RoboDK station: SETUP Fresas.rdk

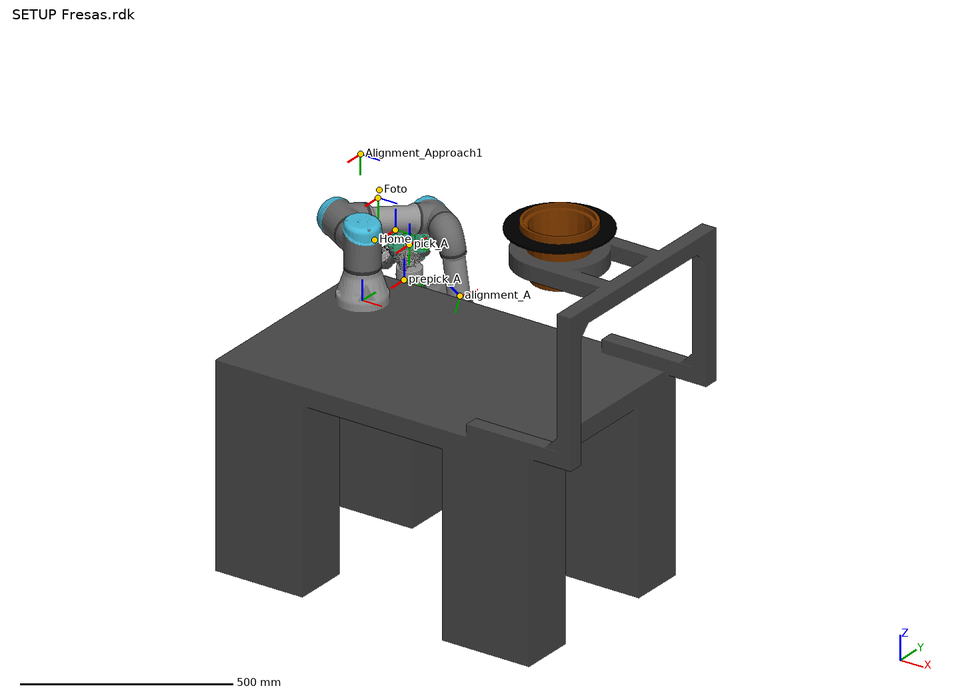
[picture v0: the station drawn from its stored meshes, robots at their saved joint values, targets as dots, program paths as lines]
Station SETUP Fresas (saved by RoboDK 5.9.2). Poses are relative to the parent item; angles as X-Y-Z fixed-axis rotations.
Station parameters (name, value as stored): RECORD_READY, 1, RECORD_ACKNOWLEDGE, 0, CollisionFreeMoveJ, None, CollisionFreeMoveL, None, PathPlanningMaxTime, 5000, PathPlanningMaxIterations, 1000
  - object Mesa SetUp v1 at (600, -20, 0) mm, size 900 x 600 x 550 mm, geometry from Mesa SetUp v1.step
  - frame UR3e Base at (700, 440, 50) mm
    - robot UR3e: 6 axes, payload 3 kg, reach 500 mm, repeatability 0.03 mm, weight 11 kg
        modified DH rows (alpha deg, a mm, theta deg, d mm): 0, 0, 0, 151.9; 90, 0, 180, 0; 0, 243.55, 0, 0; 0, 213.2, 0, 131.05; -90, 0, 0, 85.35; 90, 0, 180, 92.1
        joint limits [-360, -180, -360, -360, -360, -360] to [360, 20, 360, 360, 360, 360]; home [0, -90, -90, 0, 90, 0]; saved at [239.705, 9.056, 73.773, 7.171, -90, -59.705]
      - tool grMK2_betaMK2_asm v6, TCP at (0, 0, 57) mm, size 118.1 x 111.3 x 125.7 mm
      - tool Realsense RGB, TCP at (-11.08, -53.4, 24.76) mm, rotated rx -10 ry 0 rz 0 deg
    - target Home (joint target) at (127.85, -131.05, 246.35) mm, rotated rx -180 ry 0 rz -180 deg; joints [0, -90, -90, 90, -90, -90] of UR3e
    - target Foto (joint target) at (140.09, -131.05, 380) mm, rotated rx -80 ry 0 rz -90 deg; joints [0, -32.82, -150.904, 13.724, 90, 0] of UR3e
    - frame Prepick_plane at (200, -150, 300) mm, rotated rx 0 ry 0 rz -90 deg
      - target Prepick_plane (joint target) at (0, 0, 0) mm; joints [-5.255, -119.46, -148.452, -2.088, -90, -174.745] of UR3e
    - frame Alignment_Approach1 at (100, -150, 470) mm, rotated rx -90 ry 0 rz -90 deg
      - target Alignment_Approach1 (joint target) at (0, 0, 0) mm; joints [15.744, -17.994, -114.376, -47.63, 74.256, 0] of UR3e
    - frame Alignment_Approach2 at (150, -150, 370) mm, rotated rx -90 ry 0 rz -90 deg
      - target Alignment_Approach2 (Cartesian target) at (0, 0, 0) mm; joints [29.458, -1.123, -141.988, -36.888, 60.542, 0] of UR3e
    - target alignment_A (Cartesian target) at (144.6, 193.87, -25.91) mm, rotated rx -70.14 ry 0.6 rz 76.53 deg; joints [60.185, -57.99, -37.957, -95.541, -60.683, 5.683] of UR3e
    - frame alignment_A_frame at (144.6, 193.87, -25.91) mm, rotated rx -70.14 ry 0.6 rz 76.53 deg
    - target prepick_A (Cartesian target) at (-38.34, 226.05, -47.38) mm, rotated rx 0 ry 0 rz -90 deg; joints [60.185, -57.99, -37.957, -95.541, -60.683, 5.683] of UR3e
    - frame prepick_A_frame at (-38.34, 226.05, -47.38) mm, rotated rx 0 ry 0 rz -90 deg
    - target pick_A (Cartesian target) at (-21.45, 223.06, 51.13) mm, rotated rx 0 ry 0 rz -90 deg; joints [60.185, -57.99, -37.957, -95.541, -60.683, 5.683] of UR3e
    - frame pick_A_frame at (-21.45, 223.06, 51.13) mm, rotated rx 0 ry 0 rz -90 deg
    - target post_pick_detach_A (Cartesian target) at (-21.45, 223.06, 51.13) mm, rotated rx -90.14 ry 0.6 rz 76.53 deg; joints [239.705, 9.056, 73.773, 7.171, -90, -59.705] of UR3e
    - frame post_pick_detach_A_frame at (-21.45, 223.06, 51.13) mm, rotated rx -90.14 ry 0.6 rz 76.53 deg
  - object Set Up Fresas YEA v3 at (1570, 280, 60) mm, rotated rx 90 ry 0 rz 180 deg, size 373.6 x 472 x 595 mm, geometry from Set Up Fresas YEA v3.step
  - Python program Giro Brida (listed below)
  - Python program Giro colisiones (listed below)
  - Python program Prog6 (listed below)
  - Python program Hand_Eye_acquisition (listed below)
  - Python program Camera_Live_Stream (listed below)
  - Python program Camera_calibration (listed below)
  - Python program Hand_Eye_calibration (listed below)
  - camera Cámara1

--- Python program Giro Brida ---
from robolink import *    # API de RoboDK
from robodk import *      # Funciones matemáticas
import time
import math
import copy
import sys

# Conexión a RoboDK
RDK = Robolink()

# Intentar seleccionar el robot (usa nombre o el robot activo si '' )
robot = RDK.Item('UR3e', ITEM_TYPE_ROBOT)
if not robot.Valid():
    robot = RDK.Item('', ITEM_TYPE_ROBOT)  # fallback: robot activo
    if not robot.Valid():
        raise Exception("No se encontró ningún robot activo. Revisa el nombre o selecciona el robot en RoboDK.")

# Obtener joints crudos
j_raw = robot.Joints()

# --- Aplanar / normalizar la estructura de joints a una lista de floats ---
def normalize_joints(j):
    # Si el objeto tiene método .list() (tipo Mat), usarlo
    try:
        if hasattr(j, 'list'):
            jl = j.list()
            # jl puede ser ya lista de floats o lista dentro de lista
            if len(jl) == 1 and isinstance(jl[0], (list, tuple)):
                return list(jl[0])
            return list(jl)
    except Exception:
        pass

    # Si es iterable (tuple/list) intentar convertir y aplanar un nivel
    try:
        jl = list(j)
        if len(jl) == 1 and isinstance(jl[0], (list, tuple)):
            return list(jl[0])
        return jl
    except Exception:
        return []

joints_ini = normalize_joints(j_raw)

print("Estructura cruda de joints:", j_raw)
print("Joints normalizados:", joints_ini)

# Comprobar que hay al menos 6 articulaciones
if len(joints_ini) < 6:
    raise Exception(f"Se esperaban al menos 6 valores de articulación pero se obtuvieron {len(joints_ini)}. Imprime la salida para depurar.")

# Parámetros
amplitud = math.radians(14400)   # ±45° desde la posición inicial de J6
pasos = 180                   # pasos por medio ciclo (más = más suave)
pausa = 0.01                  # segundos entre pasos
vueltas = 4                   # número de ciclos ida+vuelta

j6_base = joints_ini[5]

print(f"J6 base = {math.degrees(j6_base):.2f}°  (valor en rad: {j6_base})")

# Ejecutar giros seguros (ida y vuelta) 4 veces
for v in range(vueltas):
    # IDA: 0 -> +amplitud -> 0 (sinusoidal)
    for i in range(pasos + 1):
        frac = i / float(pasos)
        delta = amplitud * math.sin(math.pi * frac)     # 0 -> +amplitud -> 0
        target = copy.copy(joints_ini)
        target[5] = j6_base + delta
        robot.setJoints(target)
        # opcional: forzar render si RoboDK no actualiza visual (descomenta si hace falta)
        # RDK.Render(0)
        if i % (pasos // 6 if pasos >= 6 else 1) == 0:
            print(f"[V{v+1} IDA] step {i}/{pasos} -> J6={math.degrees(target[5]):.2f}°")
        time.sleep(pausa)

    # VUELTA: 0 -> -amplitud -> 0
    for i in range(pasos + 1):
        frac = i / float(pasos)
        delta = -amplitud * math.sin(math.pi * frac)    # 0 -> -amplitud -> 0
        target = copy.copy(joints_ini)
        target[5] = j6_base + delta
        robot.setJoints(target)
        # RDK.Render(0)
        if i % (pasos // 6 if pasos >= 6 else 1) == 0:
            print(f"[V{v+1} VUELTA] step {i}/{pasos} -> J6={math.degrees(target[5]):.2f}°")
        time.sleep(pausa)

# Regresar exactamente a la posición inicial
robot.MoveJ(joints_ini)
print("Hecho: regresado a la posición inicial.")

--- Python program Giro colisiones ---
from robolink import *
from robodk import *
import math
import time
import copy

# Conectar con RoboDK
RDK = Robolink()
robot = RDK.Item('UR3e', ITEM_TYPE_ROBOT)
if not robot.Valid():
    robot = RDK.Item('', ITEM_TYPE_ROBOT)
    if not robot.Valid():
        raise Exception("No se encontró ningún robot activo")

# Activar detección de colisiones
RDK.setCollisionActive(True)

# Guardar posición inicial
joints_ini = list(robot.Joints())
j6_base = joints_ini[5]

# Parámetros de giro
vueltas = 4
pasos = 180
pausa = 0.01
amplitud = math.radians(360)  # 1 vuelta por ciclo

# Objetos a considerar para colisión (la maceta y la cámara)
maceta = RDK.Item('Set Up Fresas YEA v3')          # Ajusta el nombre exacto
camara = RDK.Item('gripper_beta_assembly v23')          # Ajusta el nombre exacto
objetos_colision = [maceta, camara]

# Función para checar colisiones
def check_collision(joints):
    robot.setJoints(joints, True)   # Posición temporal para chequeo
    col = robot.CheckCollision(objetos_colision)
    return col

# Giro con detección de colisiones
for v in range(vueltas):
    # IDA
    for i in range(pasos + 1):
        delta = amplitud * math.sin(math.pi * i / pasos)
        target = copy.copy(joints_ini)
        target[5] = j6_base + delta

        if check_collision(target):
            print(f"⚠ Colisión detectada en vuelta {v+1}, paso {i}")
            break  # detener movimiento si hay colisión

        robot.setJoints(target)
        RDK.Render(0)
        time.sleep(pausa)

    # VUELTA
    for i in range(pasos + 1):
        delta = -amplitud * math.sin(math.pi * i / pasos)
        target = copy.copy(joints_ini)
        target[5] = j6_base + delta

        if check_collision(target):
            print(f"⚠ Colisión detectada en vuelta {v+1} (regreso), paso {i}")
            break

        robot.setJoints(target)
        time.sleep(pausa)

# Regresar a la posición inicial
robot.MoveJ(joints_ini)
print("✅ Giro terminado, regresado a la posición inicial.")

--- Python program Prog6 ---
from robodk.robolink import *      # API de RoboDK
from robodk import robomath
import random

# --------------------------------------
# Parámetros principales
NUM_POSITIONS = 40
DELTA_DEGREES = 180   # variación máxima de cada junta (± grados)
ROBOT_NAME = "UR3e"  # nombre del robot en RoboDK
RECORD_READY = 'RECORD_READY'
MIN_DIFF_DEG = 5     # diferencia mínima entre posiciones (grados)
# --------------------------------------

# Conexión con RoboDK
RDK = Robolink()
robot = RDK.Item(ROBOT_NAME, ITEM_TYPE_ROBOT)

if not robot.Valid():
    raise Exception("No se encontró el robot en la estación RoboDK")

# Pose inicial del robot
current_joints = robot.Joints()

# Función para verificar que dos posiciones no sean casi iguales
def is_too_close(j1, j2, tol_deg=MIN_DIFF_DEG):
    for a, b in zip(j1, j2):
        if abs(a - b) > tol_deg * robomath.pi/180:  # pasar a radianes
            return False
    return True

# Generar configuraciones aleatorias únicas
joint_positions = []
while len(joint_positions) < NUM_POSITIONS:
    new_joints = current_joints.tolist()
    for j in range(len(new_joints)):
        delta = random.uniform(-DELTA_DEGREES, DELTA_DEGREES) * robomath.pi/180
        new_joints[j] += delta

    # Revisar que no esté repetida o muy parecida a otra
    if not any(is_too_close(new_joints, jp) for jp in joint_positions):
        joint_positions.append(new_joints)

print(f"Se generaron {len(joint_positions)} posiciones únicas")

# Mover el robot a las posiciones aleatorias y cambiar RECORD_READY
for i, joints in enumerate(joint_positions):
    try:
        print(f"Moviendo a posición {i+1}/{NUM_POSITIONS}")
        robot.MoveJ(joints)   # Movimiento en espacio articular

        # Señalizar que la posición está lista
        RDK.setParam(RECORD_READY, 1)

        # Esperar a que la otra parte procese la señal
        while int(RDK.getParam('RECORD_ACKNOWLEDGE')) != 1:
            robomath.pause(0.05)

        # Resetear acknowledge para la próxima iteración
        RDK.setParam('RECORD_ACKNOWLEDGE', 0)
        RDK.setParam(RECORD_READY, 0)

    except Exception as e:
        print(f"Error en la posición {i+1}: {e}")

print(f"Proceso terminado: {NUM_POSITIONS} movimientos completados")

--- Python program Hand_Eye_acquisition ---
# Type help("robolink") or help("robodk") for more information
# Press F5 to run the script
# Documentation: https://robodk.com/doc/en/RoboDK-API.html
# Reference:     https://robodk.com/doc/en/PythonAPI/index.html
#
# Utility script to perform hand-eye calibration on a 2D camera.
# This script can be use for eye-in-hand or eye-to-hand calibrations.
# Dynamically record the robot pose and save the camera image on disk for later processing.
# This script is running in a separate thread and a main program request punctual recordings through an handshake.

from robodk import robolink  # RoboDK API
from robodk import robomath  # Robot toolbox

# Uncomment these lines to automatically install the dependencies using pip
# robolink.import_install('cv2', 'opencv-contrib-python==4.5.*')
# robolink.import_install('numpy')
import cv2 as cv
import numpy as np
from pathlib import Path
import json
from enum import Enum
import time


#--------------------------------------
# This script supports RoboDK virtual/simulated cameras, and USB devices (as supported by OpenCV)
# You can add your own implementation to retrieve images from any camera, such as a Cognex Insight, SICK, etc.
class CameraTypes(Enum):
    ROBODK_SIMULATED = 0
    OPENCV_USB = 1


RECORD_ROBOT = True  # Record the robot pose on disk
RECORD_CAMERA = True  # Record the camera image on disk
RECORD_FOLDER = 'Hand-Eye-Data'  # Default folder to save recordings, relative to the station folder

CAMERA_TYPE = CameraTypes.ROBODK_SIMULATED  # Camera type to be used
CAMERA_ROBODK_NAME = 'Cámara1'  # [Optional] Default name to use for the RoboDK camera
ROBOT_NAME = 'UR3e'  # [Optional] Default name to use for the robot

# Station variables shared with the main program to interact with this script
RECORD_READY = 'RECORD_READY'  # Set this true in the main program when the robot is in position and the the script is allowed to record the robot and the image
RECORD_ACKNOWLEDGE = 'RECORD_ACKNOWLEDGE'  # Set this true in this script when the record is complete
RECORD_STOP = 'RECORD_STOP'  # Request to stop the script by the main program


#--------------------------------------
def get_robot(RDK: robolink.Robolink, robot_name: str):

    # Retrieve the robot
    robot_item = None
    if robot_name:
        robot_item = RDK.Item(robot_name, robolink.ITEM_TYPE_ROBOT)
        if not robot_item.Valid():
            robot_name = ''

    if not robot_name:
        robot_item = RDK.ItemUserPick("Select the robot for hand-eye", robolink.ITEM_TYPE_ROBOT)
        if not robot_item.Valid():
            raise

    return robot_item


def get_camera_handle(camera_type: CameraTypes, camera_name: str, RDK: robolink.Robolink):

    if camera_type == CameraTypes.ROBODK_SIMULATED:

        # Retrieve the RoboDK camera by name
        camera_item = None
        if camera_name:
            camera_item = RDK.Item(camera_name, robolink.ITEM_TYPE_CAMERA)
            if not camera_item.Valid():
                camera_name = ''

        if not camera_name:
            camera_item = RDK.ItemUserPick("Select the camera for hand-eye", robolink.ITEM_TYPE_CAMERA)
            if not camera_item.Valid():
                raise

        # Ensure the preview window in RoboDK is open
        if camera_item.setParam('Open') != '1':
            camera_item.setParam('Open', 1)
            robomath.pause(0.1)

        return camera_item

    elif camera_type == CameraTypes.OPENCV_USB:
        return cv.VideoCapture(0, cv.CAP_ANY)  # More information on supported devices here: https://docs.opencv.org/4.x/d8/dfe/classcv_1_1VideoCapture.html#aabce0d83aa0da9af802455e8cf5fd181

    return None


def record_camera(camera_type: CameraTypes, camera_handle, filename: str):
    if camera_type == CameraTypes.ROBODK_SIMULATED:
        record_robodk_camera(filename, camera_handle)

    elif camera_type == CameraTypes.OPENCV_USB:
        record_opencv_camera(filename, camera_handle)


def record_robodk_camera(filename: str, camera_item: robolink.Item):

    # Retrieve the image by socket
    bytes_img = camera_item.RDK().Cam2D_Snapshot('', camera_item)
    nparr = np.frombuffer(bytes_img, np.uint8)
    img = cv.imdecode(nparr, cv.IMREAD_COLOR)

    # Save the image on disk as a grayscale image
    cv.imwrite(filename, cv.cvtColor(img, cv.COLOR_RGB2GRAY))


def record_opencv_camera(filename: str, capture: cv.VideoCapture):

    # Retrieve image
    success, img = capture.read()
    if not success:
        raise

    # Save the image on disk as a grayscale image
    cv.imwrite(filename, cv.cvtColor(img, cv.COLOR_RGB2GRAY))


def record_robot(robot_item: robolink.Item, filename: str):

    # Retrieve the required information for hand-eye
    robot_data = {}
    robot_data['joints'] = robot_item.Joints().tolist()
    robot_data['pose_flange'] = robomath.Pose_2_TxyzRxyz(robot_item.SolveFK(robot_item.Joints()))

    # Save it on disk as a JSON
    # You can also provide another format, like YAML
    with open(filename, 'w') as f:
        json.dump(robot_data, f, indent=2)


def runmain():

    RDK = robolink.Robolink()

    # Retrieve the camera and robot
    camera_handle = get_camera_handle(CAMERA_TYPE, CAMERA_ROBODK_NAME, RDK)
    print ("Camera name:" + camera_handle.Name())
    robot_item = get_robot(RDK, ROBOT_NAME)
    print ("Robot name:" + robot_item.Name())

    # Retrieve the folder to save the data
    record_folder = Path(RDK.getParam(robolink.PATH_OPENSTATION)) / RECORD_FOLDER
    record_folder.mkdir(exist_ok=True, parents=True)
    print ("Folder ok")
    # This script does not delete the previous run if the folder is not empty
    # If the folder is not empty, retrieve the next ID
    id = 0
    ids = sorted([int(x.stem) for x in record_folder.glob('*.png') if x.stem.isdigit()])
    if ids:
        id = ids[-1] + 1

    # Start the main loop, and wait for requests
    RDK.setParam(RECORD_READY, 0)

    while True:
        time.sleep(0.01)

        # Read the requests set by the main program
        ready = int(RDK.getParam(RECORD_READY)or 0) == 1
        stop = int(RDK.getParam(RECORD_STOP)or 0) == 1
        if stop:
            break

        if not ready:
            continue

        # Process the requests
        if RECORD_CAMERA:
            img_filename = Path(f'{record_folder.as_posix()}/{id}.png')
            record_camera(CAMERA_TYPE, camera_handle, img_filename.as_posix())

        if RECORD_ROBOT:
            robot_filename = Path(f'{record_folder.as_posix()}/{id}.json')
            record_robot(robot_item, robot_filename.as_posix())

        id += 1

        print(img_filename)
        print(robot_filename)

        # Inform the main program that we have completed the request
        RDK.setParam(RECORD_ACKNOWLEDGE, 1)
        RDK.setParam(RECORD_READY, 0)


if __name__ == '__main__':
    runmain()

--- Python program Camera_Live_Stream ---
# Type help("robodk.robolink") or help("robodk.robomath") for more information
# Press F5 to run the script
# Documentation: https://robodk.com/doc/en/RoboDK-API.html
# Reference:     https://robodk.com/doc/en/PythonAPI/index.html
#
# This example demonstrates some of the basic functionalities to handle 2D cameras using the RoboDK API for Python.
# It creates/reuses an existing camera, set its parameters, get the image using two different methods and display it to the user as a live stream.
# This is a great starting point for your computer vision algorithms.
#

from robodk import robolink  # RoboDK API
from robodk import robomath  # Robot toolbox
RDK = robolink.Robolink()

# OpenCV is an open source Computer Vision toolkit, which you can use to filter and analyse images
robolink.import_install('cv2', 'opencv-python', RDK)
robolink.import_install('numpy', RDK)
import numpy as np
import cv2 as cv

CAM_NAME = 'Cámara 1'
CAM_PARAMS = 'SIZE=640x480' # For more options, see https://robodk.com/doc/en/PythonAPI/robodk.html#robodk.robolink.Robolink.Cam2D_Add
WINDOW_NAME = 'My Camera Feed'

#----------------------------------
# Get the camera item
cam_item = RDK.Item(CAM_NAME, robolink.ITEM_TYPE_CAMERA)
if not cam_item.Valid():
    cam_item = RDK.Cam2D_Add(RDK.AddFrame(CAM_NAME + ' Frame'), CAM_PARAMS)
    cam_item.setName(CAM_NAME)
cam_item.setParam('Open', 1)

#----------------------------------
# Create a live feed
while cam_item.setParam('isOpen') == '1':

    #----------------------------------
    # Method 1: Get the camera image, by socket
    img_socket = None
    bytes_img = RDK.Cam2D_Snapshot('', cam_item)
    if isinstance(bytes_img, bytes) and bytes_img != b'':
        nparr = np.frombuffer(bytes_img, np.uint8)
        img_socket = cv.imdecode(nparr, cv.IMREAD_COLOR)
    if img_socket is None:
        break

    #----------------------------------
    # Method 2: Get the camera image, from disk
    img_png = None
    import tempfile
    with tempfile.TemporaryDirectory(prefix='robodk_') as td:
        tf = td + '/temp.png'
        if RDK.Cam2D_Snapshot(tf, cam_item) == 1:
            img_png = cv.imread(tf)
    if img_png is None:
        break

    #----------------------------------
    # Show it to the world!
    cv.imshow(WINDOW_NAME, img_socket)
    key = cv.waitKey(1)
    if key == 27:
        break  # User pressed ESC, exit
    if cv.getWindowProperty(WINDOW_NAME, cv.WND_PROP_VISIBLE) < 1:
        break  # User killed the main window, exit

# Close the preview and the camera. Ensure you call cam_item.setParam('Open', 1) before reusing a camera!
cv.destroyAllWindows()
RDK.Cam2D_Close(cam_item)

--- Python program Camera_calibration ---
# Type help("robolink") or help("robodk") for more information
# Press F5 to run the script
# Documentation: https://robodk.com/doc/en/RoboDK-API.html
# Reference:     https://robodk.com/doc/en/PythonAPI/index.html
#
# Find a camera intrinsic and extrinsic properties using a chessboard and a series of images.
# More details on camera calibration: https://docs.opencv.org/master/dc/dbb/tutorial_py_calibration.html
# You can print this board in letter format: https://github.com/opencv/opencv/blob/master/doc/pattern.png

from robodk.robolink import *
from robodk.robodialogs import *
import cv2 as cv
import numpy as np
import glob

#----------------------------------------------
# You can edit these settings for your board
SQUARES_X = 10  # number of squares along the X axis
SQUARES_Y = 7  # number of squares along the Y axis
PATTERN = (SQUARES_X - 1, SQUARES_Y - 1)
SQUARE_LENGTH = 23.0  # mm, length of one square

#----------------------------------------------
# Get the images
images_dir = getSaveFolder(popup_msg='Select the directory of the images')
images = glob.glob('%s/*.png' % images_dir) + glob.glob('%s/*.jpg' % images_dir)

#----------------------------------------------
# Parse the images
frame_size = None
obj_points = []  # 3D points in real world space
img_points = []  # 2D points in image plane.
objp = np.zeros((PATTERN[0] * PATTERN[1], 3), np.float32)  # object points (0,0,0), (1,0,0), (2,0,0) ....,(8,5,0)
objp[:, :2] = np.mgrid[0:PATTERN[0], 0:PATTERN[1]].T.reshape(-1, 2) * SQUARE_LENGTH

for image in images:
    # Read the image as grayscale
    img = cv.imread(image)
    gray = cv.cvtColor(img, cv.COLOR_BGR2GRAY)
    frame_size = gray.shape[::-1]

    # Find the chessboard corners
    ret, corners = cv.findChessboardCorners(gray, PATTERN, None)

    # If found, add object points, image points (after refining them)
    if ret == True:
        rcorners = cv.cornerSubPix(gray, corners, (11, 11), (-1, -1), (cv.TERM_CRITERIA_EPS + cv.TERM_CRITERIA_MAX_ITER, 30, 0.001))
        img_points.append(rcorners)
        obj_points.append(objp)

        # Draw and display the corners
        cv.drawChessboardCorners(img, PATTERN, rcorners, ret)
        cv.imshow('Original image', img)
        cv.waitKey(250)

cv.destroyAllWindows()

#----------------------------------------------
# Get the calibrated camera parameters
rms_err, calib_mtx, dist_coeffs, rvecs, tvecs = cv.calibrateCamera(obj_points, img_points, frame_size, None, None)
print('Overall RMS re-projection error: %0.3f' % rms_err)

#----------------------------------------------
# Save the parameters
file = getSaveFileName(strfile='RoboDK-Camera-Settings.yaml', defaultextension='.yaml', filetypes=[('YAML files', '.yaml')])
cv_file = cv.FileStorage(file, cv.FILE_STORAGE_WRITE)
if not cv_file.isOpened():
    raise Exception('Failed to save calibration file')
cv_file.write("camera_matrix", calib_mtx)
cv_file.write("dist_coeff", dist_coeffs)
cv_file.write("camera_size", frame_size)
cv_file.release()

--- Python program Hand_Eye_calibration ---
# Type help("robolink") or help("robodk") for more information
# Press F5 to run the script
# Documentation: https://robodk.com/doc/en/RoboDK-API.html
# Reference:     https://robodk.com/doc/en/PythonAPI/index.html
#
# Perform hand-eye calibration with recorded robot poses and 2D images from disk.
# - Requires at least 8 different poses at different orientations/distances of a chessboard or charucoboard.
# - Requires a calibrated camera (known intrinsic parameters, including distortion), which can also be performed from local images.
#
# You can find the board used in this example here:
# https://docs.opencv.org/4.x/charucoboard.png
#

from robodk import robolink  # RoboDK API
from robodk import robomath  # Robot toolbox
from robodk import robodialogs  # Dialogs

# Uncomment these lines to automatically install the dependencies using pip
# robolink.import_install('cv2', 'opencv-contrib-python==4.5.*')
# robolink.import_install('numpy')
import cv2 as cv
import numpy as np
import json
from pathlib import Path
from enum import Enum


#--------------------------------------
# This scripts supports chessboard (checkerboard) and ChAruCo board as calibration objects.
# You can add your own implementation (such as dot patterns).
class MarkerTypes(Enum):
    CHESSBOARD = 0
    CHARUCOBOARD = 1


# The camera intrinsic parameters can be performed with the same board as the Hand-eye
INTRINSIC_FOLDER = 'Hand-Eye-Data'  # Default folder to load images for the camera calibration, relative to the station folder
HANDEYE_FOLDER = 'Hand-Eye-Data'  # Default folder to load robot poses and images for the hand-eye calibration, relative to the station folder

# Camera intrinsic calibration board parameters
# You can find this chessboard here: https://docs.opencv.org/4.x/charucoboard.png
INTRINSIC_BOARD_TYPE = MarkerTypes.CHESSBOARD
INTRINSIC_CHESS_SIZE = (7, 10)  # X/Y
INTRINSIC_SQUARE_SIZE = 25  # mm
INTRINSIC_MARKER_SIZE = 21  # mm

# Hand-eye calibration board parameters
# You can find this charucoboard here: https://docs.opencv.org/4.x/charucoboard.png
#HANDEYE_BOARD_TYPE = MarkerTypes.CHARUCOBOARD
HANDEYE_BOARD_TYPE = MarkerTypes.CHESSBOARD
HANDEYE_CHESS_SIZE = (7, 10)  # X/Y
HANDEYE_SQUARE_SIZE = 25  # mm
HANDEYE_MARKER_SIZE = 21  # mm


def pose_2_Rt(pose: robomath.Mat):
    """RoboDK pose to OpenCV pose"""
    pose_inv = pose.inv()
    R = np.array(pose_inv.Rot33())
    t = np.array(pose.Pos())
    return R, t

def Rt_2_pose(R, t):
    """
    OpenCV rotation matrix R (3x3) and translation vector t (3x1)
    -> RoboDK Pose
    """
    cam_pose = robomath.eye(4)

    # Set rotation vectors
    vx = R[:,0].flatten().tolist()
    vy = R[:,1].flatten().tolist()
    vz = R[:,2].flatten().tolist()
    cam_pose.setVX(vx)
    cam_pose.setVY(vy)
    cam_pose.setVZ(vz)

    # Set translation
    cam_pose.setPos(t.flatten().tolist())

    return cam_pose



def find_chessboard(img, mtx, dist, chess_size, squares_edge, refine=True, draw_img=True):
    """
    Detects a chessboard pattern in an image.
    """

    pattern = np.subtract(chess_size, (1, 1))  # number of corners

    # Prefer grayscale images
    _img = img
    if len(img.shape) > 2:
        _img = cv.cvtColor(img, cv.COLOR_RGB2GRAY)

    # Find the chessboard's corners
    success, corners = cv.findChessboardCorners(_img, pattern)
    if not success:
        raise Exception("No chessboard found")

    # Refine
    if refine:
        criteria = (cv.TERM_CRITERIA_EPS + cv.TERM_CRITERIA_MAX_ITER, 30, 0.001)
        search_size = (11, 11)
        zero_size = (-1, -1)
        corners = cv.cornerSubPix(_img, corners, search_size, zero_size, criteria)

    if draw_img is not None:
        cv.drawChessboardCorners(draw_img, pattern, corners, success)

    # Find the camera pose. Only available with the camera matrix!
    if mtx is None or dist is None:
        return corners, None, None

    cb_corners = np.zeros((pattern[0] * pattern[1], 3), np.float32)
    cb_corners[:, :2] = np.mgrid[0:pattern[0], 0:pattern[1]].T.reshape(-1, 2) * squares_edge
    success, rvec, tvec = cv.solvePnP(cb_corners, corners, mtx, dist)
    if not success:
        raise Exception("No chessboard found")

    R_target2cam = cv.Rodrigues(rvec)[0]
    t_target2cam = tvec

    return corners, R_target2cam, t_target2cam


def find_charucoboard(img, mtx, dist, chess_size, squares_edge, markers_edge, predefined_dict=cv.aruco.DICT_6X6_100, draw_img=True) -> dict:
    """
    Detects a charuco board pattern in an image.
    """

    # Note that for chessboards, the pattern size is the number of "inner corners", while charucoboards are the number of chessboard squares

    # Charuco board and dictionary
    charuco_board = cv.aruco.CharucoBoard_create(chess_size[0], chess_size[1], squares_edge, markers_edge, cv.aruco.getPredefinedDictionary(predefined_dict))
    charuco_dict = charuco_board.dictionary

    # Find the markers first
    marker_corners, marker_ids, _ = cv.aruco.detectMarkers(img, charuco_dict, None, None, None, None)
    if marker_ids is None or len(marker_ids) < 1:
        raise Exception("No charucoboard found")

    # Then the charuco
    count, corners, ids = cv.aruco.interpolateCornersCharuco(marker_corners, marker_ids, img, charuco_board, None, None, mtx, dist, 2)  # mtx and dist are optional here
    if count < 1 or len(ids) < 1:
        raise Exception("No charucoboard found")

    if draw_img is not None:
        cv.aruco.drawDetectedCornersCharuco(draw_img, corners, ids)

    # Find the camera pose. Only available with the camera matrix!
    if mtx is None or dist is None:
        return corners, None, None

    success, rot_vec, trans_vec = cv.aruco.estimatePoseCharucoBoard(corners, ids, charuco_board, mtx, dist, None, None, False)  # mtx and dist are mandatory here
    if not success:
        raise Exception("Charucoboard pose not found")

    if draw_img is not None:
        cv.drawFrameAxes(draw_img, mtx, dist, rot_vec, trans_vec, max(1.5 * squares_edge, 5))

    R_target2cam = cv.Rodrigues(rot_vec)[0]

    return corners, R_target2cam, trans_vec


def calibrate_static(chessboard_images, board_type: MarkerTypes, chess_size, squares_edge: float, markers_edge: float, min_detect: int = -1, show_images=True):
    """
    Calibrate a camera with a chessboard or charucoboard pattern.
    """
    # Chessboard parameters
    pattern = np.subtract(chess_size, (1, 1))  # number of corners
    img_size = None

    # Find the chessboard corners
    img_corners = []

    if show_images:
        WDW_NAME = 'Chessboard'
        MAX_W, MAX_H = 640, 480
        cv.namedWindow(WDW_NAME, cv.WINDOW_NORMAL)

    for file, img in chessboard_images.items():
        # Ensure the image size is consistent
        if img_size is None:
            img_size = img.shape[:2]
        else:
            if img.shape[:2] != img_size:
                raise Exception('Camera resolution is not consistent across images!')

        # Find the chessboard corners
        draw_img = None
        if show_images:
            draw_img = cv.cvtColor(img, cv.COLOR_GRAY2RGB)
        try:
            if board_type == MarkerTypes.CHESSBOARD:
                corners, _, _ = find_chessboard(img, mtx=None, dist=None, chess_size=chess_size, squares_edge=squares_edge, draw_img=draw_img)
            else:
                corners, _, _ = find_charucoboard(img, mtx=None, dist=None, chess_size=chess_size, squares_edge=squares_edge, markers_edge=markers_edge, draw_img=draw_img)
        except:
            print(f'Unable to find chessboard in {file}!')
            continue

        if show_images:
            cv.imshow(WDW_NAME, draw_img)
            cv.resizeWindow(WDW_NAME, MAX_W, MAX_H)
            cv.waitKey(500)
        img_corners.append(corners)

        # Check if we processed enough images
        if min_detect > 0 and len(img_corners) >= min_detect:
            break

    if show_images:
        cv.destroyAllWindows()

    if len(img_corners) < 3 or min_detect > 0 and len(img_corners) < min_detect:
        raise Exception('Not enough detections!')

    # Calibrate the camera
    # Create a flat chessboard representation of the corners
    cb_corners = np.zeros((pattern[0] * pattern[1], 3), np.float32)
    cb_corners[:, :2] = np.mgrid[0:pattern[0], 0:pattern[1]].T.reshape(-1, 2) * squares_edge

    h, w = img_size
    rms_err, mtx, dist, rot_vecs, trans_vecs = cv.calibrateCamera([cb_corners for i in range(len(img_corners))], img_corners, (w, h), None, None)
    return mtx, dist, (w, h)


def calibrate_handeye(robot_poses, chessboard_images, camera_matrix, camera_distortion, board_type: MarkerTypes, chess_size, squares_edge: float, markers_edge: float, show_images=True):
    """
    Calibrate a camera mounted on a robot arm using a list of robot poses and a list of images for each pose.
    The robot pose should be at the flange (remove .PoseTool) unless you have a calibrated tool.
    """
    # https://docs.opencv.org/4.x/d9/d0c/group__calib3d.html#gaebfc1c9f7434196a374c382abf43439b

    # Rotation part extracted from the homogeneous matrix that transforms a point expressed in the gripper frame to the robot base frame (bTg).
    # This is a vector (vector<Mat>) that contains the rotation, (3x3) rotation matrices or (3x1) rotation vectors, for all the transformations from gripper frame to robot base frame.
    R_gripper2base_list = []

    # Translation part extracted from the homogeneous matrix that transforms a point expressed in the gripper frame to the robot base frame (bTg).
    # This is a vector (vector<Mat>) that contains the (3x1) translation vectors for all the transformations from gripper frame to robot base frame.
    t_gripper2base_list = []

    # Rotation part extracted from the homogeneous matrix that transforms a point expressed in the target frame to the camera frame (cTt).
    # This is a vector (vector<Mat>) that contains the rotation, (3x3) rotation matrices or (3x1) rotation vectors, for all the transformations from calibration target frame to camera frame.
    R_target2cam_list = []

    # Rotation part extracted from the homogeneous matrix that transforms a point expressed in the target frame to the camera frame (cTt).
    # This is a vector (vector<Mat>) that contains the (3x1) translation vectors for all the transformations from calibration target frame to camera frame.
    t_target2cam_list = []

    if show_images:
        WDW_NAME = 'Charucoboard'
        #WDW_NAME = 'Chessboard'
        MAX_W, MAX_H = 640, 480
        cv.namedWindow(WDW_NAME, cv.WINDOW_NORMAL)

    for i in chessboard_images.keys():
        robot_pose = robot_poses[i]
        image = chessboard_images[i]
        draw_img = None
        if show_images:
            draw_img = cv.cvtColor(image, cv.COLOR_GRAY2RGB)
        try:
            if board_type == MarkerTypes.CHESSBOARD:
                _, R_target2cam, t_target2cam = find_chessboard(image, camera_matrix, camera_distortion, chess_size, squares_edge, draw_img=draw_img)
            else:
                _, R_target2cam, t_target2cam = find_charucoboard(image, camera_matrix, camera_distortion, chess_size, squares_edge, markers_edge, draw_img=draw_img)
        except:
            print(f'Unable to find chessboard in {i}!')
            continue

        if show_images:
            cv.imshow(WDW_NAME, draw_img)
            cv.resizeWindow(WDW_NAME, MAX_W, MAX_H)
            cv.waitKey(500)

        R_target2cam_list.append(R_target2cam)
        t_target2cam_list.append(t_target2cam)

        R_gripper2base, t_gripper2base = pose_2_Rt(robot_pose)
        R_gripper2base_list.append(R_gripper2base)
        t_gripper2base_list.append(t_gripper2base)

    if show_images:
        cv.destroyAllWindows()

    R_cam2gripper, t_cam2gripper = cv.calibrateHandEye(R_gripper2base_list, t_gripper2base_list, R_target2cam_list, t_target2cam_list)
    return Rt_2_pose(R_cam2gripper, t_cam2gripper)


def runmain():
    #------------------------------------------------------
    # Calibrate the camera intrinsic parameters
    # 1. Print a chessboard, measure it using a caliper
    # 2. Mount the camera statically, take a series of images of the chessboard at different distance, orientation, offset, etc.
    # 3. Calibrate the camera using the images (can be done offline)
    #
    #
    # Calibrate the camera location (hand-eye)
    # 4. Create a robot program in RoboDK that moves the robot around a static chessboard at different distance, orientation, offset, etc.
    # 5. At each position, record the robot pose (robot.Pose(), or robot.Joints() even) and take a screenshot with the camera
    # 6. Use the robot poses and the images to calibrate the camera location
    #
    #
    # Good to know
    # - You can retrieve the camera image live with OpenCV using cv.VideoCapture(0, cv.CAP_DSHOW)
    # - You can load/save images with OpenCV using cv.imread(filename) and cv.imwrite(filename, img)
    # - You can save your calibrated camera parameters with JSON, i.e. print(json.dumps({"mtx":mtx, "dist":dist}))
    #
    #------------------------------------------------------

    RDK = robolink.Robolink()

    #------------------------------------------------------
    # Calibrate a camera using local images of chessboards, retrieves the camera intrinsic parameters
    # Get the input folder
    intrinsic_folder = Path(RDK.getParam(robolink.PATH_OPENSTATION)) / INTRINSIC_FOLDER
    if not intrinsic_folder.exists():
        intrinsic_folder = robodialogs.getSaveFolder(intrinsic_folder.as_posix(), 'Select the directory containing the images (.png) for the camera intrinsic calibration')
        if not intrinsic_folder:
            raise
        intrinsic_folder = Path(intrinsic_folder)

    # Retrieve the images
    image_files = sorted(intrinsic_folder.glob('*.png'))
    images = {int(image_file.stem): cv.imread(image_file.as_posix(), cv.IMREAD_GRAYSCALE) for image_file in image_files}

    # Perform the image calibration
    mtx, dist, size = calibrate_static(images, INTRINSIC_BOARD_TYPE, INTRINSIC_CHESS_SIZE, INTRINSIC_SQUARE_SIZE, INTRINSIC_MARKER_SIZE, min_detect=-1)
    print(f'Camera matrix:\n{mtx}\n')
    print(f'Distortion coefficient:\n{dist}\n')
    print(f'Camera resolution:\n{size}\n')

    #------------------------------------------------------
    # Load images and robot poses to calibrate hand-eye camera
    # Get the input folder
    handeye_folder = Path(RDK.getParam(robolink.PATH_OPENSTATION)) / HANDEYE_FOLDER
    if not handeye_folder.exists():
        handeye_folder = robodialogs.getSaveFolder('Select the directory of the images (.png) and robot poses (.json) for hand-eye calibration')
        if not handeye_folder:
            raise
        handeye_folder = Path(handeye_folder)

    # Retrieve the images and robot poses
    image_files = sorted(handeye_folder.glob('*.png'))
    robot_files = sorted(handeye_folder.glob('*.json'))

    images, poses, joints = {}, {}, {}
    for image_file, robot_file in zip(image_files, robot_files):
        if int(image_file.stem) != int(robot_file.stem):
            raise

        id = int(image_file.stem)

        image = cv.imread(image_file.as_posix(), cv.IMREAD_GRAYSCALE)
        images[id] = image

        with open(robot_file.as_posix(), 'r') as f:
            robot_data = json.load(f)
            joints[id] = robot_data['joints']
            poses[id] = robomath.TxyzRxyz_2_Pose(robot_data['pose_flange'])

    # Perform hand-eye calibration
    camera_pose = calibrate_handeye(poses, images, mtx, dist, HANDEYE_BOARD_TYPE, HANDEYE_CHESS_SIZE, HANDEYE_SQUARE_SIZE, HANDEYE_MARKER_SIZE)
    print(f'Camera pose (wrt to the robot flange):\n{camera_pose}')

    RDK.ShowMessage('Hand-Eye location:\n' + str(camera_pose))

    #------------------------------------------------------
    # In RoboDK, set the camera location wrt to the robot flange at that calibrated hand-eye location (use a .tool)
    tool = RDK.ItemUserPick('Select the "eye" tool to calibrate', RDK.ItemList(robolink.ITEM_TYPE_TOOL))
    if tool.Valid():
        tool.setPoseTool(camera_pose)


if __name__ == '__main__':
    runmain()
